FUNCTION_BLOCK PUBLIC EventMsg
VAR_INPUT

END_VAR
VAR_OUTPUT
END_VAR
VAR
	CfgEvent                : TcEvent;
    fbEvent                 : ADSLOGEVENT;
    bSetEvent               : BOOL;(* Rising edge sets event *)  
	bInitialize : BOOL := TRUE;
END_VAR

IF (bInitialize) THEN
	CfgEvent.Class := TCEVENTCLASS_ALARM;
	CfgEvent.Prio := 2;
	CfgEvent.Id := 1;
	CfgEvent.SourceId := 17001;
	CfgEvent.bQuitRequired := FALSE;//TRUE;
	CfgEvent.Flags := TCEVENTFLAG_LOG OR TCEVENTFLAG_SRCID OR TCEVENTFLAG_AUTOFMTALL;
	CfgEvent.StreamType := TCEVENTSTREAM_SIMPLE;
	CfgEvent.ProgId :='TcEventFormatter.TcXMLFormatter' ;
    bInitialize:= FALSE;	
END_IF

fbEvent(Event:=FALSE);

METHOD PUBLIC SendEventMsg : BOOL
VAR_INPUT
	MsgClass :		UDINT;
	EventID :		UDINT;
	SourceID : 		UDINT;
END_VAR

CfgEvent.Class := MsgClass;
CfgEvent.Id := EventID;
CfgEvent.SourceId := SourceID;
fbEvent( NETID:= '',
        PORT:= 110,
        Event:=TRUE,					//Looking for rising edge here.
        EventConfigData:= CfgEvent,        
        TMOUT:= T#3S);
fbEvent(Event:= FALSE);		// transition, if not already done to falling edge
END_METHOD

END_FUNCTION_BLOCK

(* stored: Version 1.1.0.1, ProductVersion 3.1.4020.12
   POU EventMsg: Id {fc5ade13-1038-4ae2-90bb-debf2ec12c51}, SpecialFunc None
   Method SendEventMsg: Id {f580e47c-e1a2-4452-a3d0-0b82ba5d1333} *)
